// TIA Portal V17 export
// export: Created 2025-05-22T06:01:47.0303158Z, ExportSetting WithDefaults, DisplayName Totally Integrated Automation Portal, DisplayVersion V17 Update 8, DisplayName TIA Portal Openness, DisplayVersion V17 Update 8, DisplayName TIA Portal Version Control Interface, DisplayVersion V17, DisplayName SINAMICS Startdrive Advanced, DisplayVersion V17 SP2, DisplayName SINAMICS Startdrive G110M, G120, G120C, G120D, G120P, G115D, DisplayVersion V17 SP2, DisplayName SINAMICS Startdrive G130, G150, S120, S150, SINAMICS MV, S210, DisplayVersion V17 SP2, DisplayName STEP 7 Professional, DisplayVersion V17 Update 8, DisplayName SINUMERIK ONE STEP 7 Toolbox, DisplayVersion V17 Update 12, DisplayName SINUMERIK ONE PLC Basic Program Plus, DisplayVersion V17 Update 12, DisplayName SINUMERIK 840D sl STEP 7 Toolbox, DisplayVersion V17 Update 12, DisplayName STEP 7 Safety, DisplayVersion V17 Update 6, DisplayName WinCC Advanced, DisplayVersion V17 Update 8
TYPE "ALARM"
// stored: IsFailsafeCompliant false
   STRUCT
      WRONG_TOOL_MAG_POCKET : Bool;   // WRONG TOOL FOR CURRENT MAGAZINE POCKET / WRONG TOOL MAG POCKET
      WRONG_TOOL_NAME : Bool;   // WRONG TOOL NAME
      INVALID_LINE_FOR_TOOL : Bool;   // INVALID LINE FOR TOOL
      INVALID_OPERATI_FOR_TOOL : Bool;   // INVALID OPERATION FOR TOOL / INVALID OPERATI FOR TOOL
      INVALID_MACHINE_FOR_TOOL : Bool;   // INVALID MACHINE FOR TOOL
      TOOL_NOT_DECLARED : Bool;   // TOOL NOT DECLARED ON POCKET POSITION / TOOL NOT DECLARED
      TOOL_LIFE_EXPIRED_1 : Bool;   // TOOL LIFE EXPIRED 1
      TOOL_LIFE_EXPIRED_2 : Bool;   // TOOL LIFE EXPIRED 2
      TOOL_LIFE_EXPIRED_3 : Bool;   // TOOL LIFE EXPIRED 3
      TOOL_LIFE_EXPIRED_4 : Bool;   // TOOL LIFE EXPIRED 4
      TOOL_LIFE_EXPIRED_5 : Bool;   // TOOL LIFE EXPIRED 5
      QUANTTY_GTR_TARGET_1 : Bool;   // QUANTITY GREATER THAN TARGET 1 / QUANTTY GTR TARGET 1
      QUANTTY_GTR_TARGET_2 : Bool;   // QUANTITY GREATER THAN TARGET 2 / QUANTTY GTR TARGET 2
      QUANTTY_GTR_TARGET_3 : Bool;   // QUANTITY GREATER THAN TARGET 3 / QUANTTY GTR TARGET 3
      QUANTTY_GTR_TARGET_4 : Bool;   // QUANTITY GREATER THAN TARGET 4 / QUANTTY GTR TARGET 4
      QUANTTY_GTR_TARGET_5 : Bool;   // QUANTTY GTR TARGET 5
      TOOL_LIFE_GTR_TARGET_1 : Bool;   // TOOL LIFE GREATER THAN TARGET 1 / TOOL LIFE GTR TARGET 1
      TOOL_LIFE_GTR_TARGET_2 : Bool;   // TOOL LIFE GREATER THAN TARGET 2 / TOOL LIFE GTR TARGET 2
      TOOL_LIFE_GTR_TARGET_3 : Bool;   // TOOL LIFE GREATER THAN TARGET 3 / TOOL LIFE GTR TARGET 3
      TOOL_LIFE_GTR_TARGET_4 : Bool;   // TOOL LIFE GREATER THAN TARGET 4 / TOOL LIFE GTR TARGET 4
      TOOL_LIFE_GTR_TARGET_5 : Bool;   // TOOL LIFE GTR TARGET 5
      WARNING_TL_GTR_TARGET_1 : Bool;   // WARNING TOOL GREATER THAN TARGET 1 / WARNING TL GTR TARGET 1
      WARNING_TL_GTR_TARGET_2 : Bool;   // WARNING TOOL GREATER THAN TARGET 2 / WARNING TL GTR TARGET 2
      WARNING_TL_GTR_TARGET_3 : Bool;   // WARNING TOOL GREATER THAN TARGET 3 / WARNING TL GTR TARGET 3
      WARNING_TL_GTR_TARGET_4 : Bool;   // WARNING TOOL GREATER THAN TARGET 4 / WARNING TL GTR TARGET 4
      WARNING_TL_GTR_TARGET_5 : Bool;   // WARNING TL GTR TARGET 5
      INVALID_OEM_1 : Bool;   // INVALID OEM 1
      INVALID_OEM_2 : Bool;   // INVALID OEM 2
      INVALID_OEM_3 : Bool;   // INVALID OEM 3
      INVALID_OEM_4 : Bool;   // INVALID OEM 4
      INVALID_OEM_5 : Bool;   // INVALID OEM 5
      INVALID_OEM_6 : Bool;   // INVALID OEM 6
      INVALID_OEM_7 : Bool;   // INVALID OEM 7
      INVALID_OEM_8 : Bool;   // INVALID OEM 8
      INVALID_OEM_9 : Bool;   // INVALID OEM 9
      INVALID_OEM_10 : Bool;   // INVALID OEM 10
      WRONG_DUPLO_NUM : Bool;   // WRONG DUPLO NUM
      WRONG_NUMBER_CUTTING_EDGE : Bool;   // WRONG NUMBER CUTTING EDGES / WRONG NUMBER CUTTING EDGE
      INVALID_TOOL_TYPE_1 : Bool;   // INVALID TOOL TYPE EDGE 1 / INVALID TOOL TYPE 1
      INVALID_TOOL_TYPE_2 : Bool;   // INVALID TOOL TYPE EDGE 2 / INVALID TOOL TYPE 2
      INVALID_TOOL_TYPE_3 : Bool;   // INVALID TOOL TYPE EDGE 3 / INVALID TOOL TYPE 3
      INVALID_TOOL_TYPE_4 : Bool;   // INVALID TOOL TYPE EDGE 4 / INVALID TOOL TYPE 4
      INVALID_TOOL_TYPE_5 : Bool;   // INVALID TOOL TYPE 5
      WRONG_MONITORING_TYPE : Bool;   // WRONG MONITORING TYPE
      WRONG_TOOL_LOCATION_TYPE : Bool;   // WRONG TOOL LOCATION TYPE
      WRONG_CHECK_TOOL_BROKEN : Bool;   // WRONG CHECK TOOL BROKEN
      LENGTH_OUT_TOLERANCE_1 : Bool;   // TOOL LENGTH 1 OUT OF TOLERANCE / LENGTH OUT TOLERANCE 1
      LENGTH_OUT_TOLERANCE_2 : Bool;   // TOOL LENGTH 2 OUT OF TOLERANCE / LENGTH OUT TOLERANCE 2
      LENGTH_OUT_TOLERANCE_3 : Bool;   // TOOL LENGTH 3 OUT OF TOLERANCE / LENGTH OUT TOLERANCE 3
      LENGTH_OUT_TOLERANCE_4 : Bool;   // TOOL LENGTH 4 OUT OF TOLERANCE / LENGTH OUT TOLERANCE 4
      LENGTH_OUT_TOLERANCE_5 : Bool;   // LENGTH OUT TOLERANCE 5
      RADIUS_OUT_TOLERANCE_1 : Bool;   // TOOL RADIUS 1 OUT OF TOLERANCE / RADIUS OUT TOLERANCE 1
      RADIUS_OUT_TOLERANCE_2 : Bool;   // TOOL RADIUS 2 OUT OF TOLERANCE / RADIUS OUT TOLERANCE 2
      RADIUS_OUT_TOLERANCE_3 : Bool;   // TOOL RADIUS 3 OUT OF TOLERANCE / RADIUS OUT TOLERANCE 3
      RADIUS_OUT_TOLERANCE_4 : Bool;   // TOOL RADIUS 4 OUT OF TOLERANCE / RADIUS OUT TOLERANCE 4
      RADIUS_OUT_TOLERANCE_5 : Bool;   // RADIUS OUT TOLERANCE 5
      WRONG_PITCH_1 : Bool;   // WRONG PITCH 1
      WRONG_PITCH_2 : Bool;   // WRONG PITCH 2
      TOOL_NOT_LOCKED : Bool;   // TOOL NOT LOCKED
   END_STRUCT;
END_TYPE
